FUNCTION_BLOCK TcpConnection
VAR_INPUT
END_VAR
VAR_OUTPUT
END_VAR
VAR
	fbSocketListion : FB_SocketListen;
	fbSocketAccept : FB_SocketAccept;
	fbSocketConnect : FB_SocketConnect;
	fbSocketClose : FB_SocketClose;
	fbSocketCloseAll : FB_SocketCloseAll;
	fbSocketSend : FB_SocketSend;
	fbSocketReceive : FB_SocketReceive;
	fbGetLinkStatus: FB_SocketGetLinkStatus;
	
	CurrentSocket : T_HSOCKET;
	bEstablished : BOOL;
	_HistorySocketIndex : UDINT := 0;
	_HistorySocket : ARRAY[0..HISTORYSOCKET_MAX] OF T_HSOCKET;
	
	ErrorID : UDINT;
	
END_VAR

VAR CONSTANT
	SOCKETEMPTY: T_HSOCKET 
		:= (handle := 0, 
			localAddr := (nPort := 0, sAddr := ''), 
			remoteAddr := (nPort := 0, sAddr := ''));
	HISTORYSOCKET_MAX: UDINT  := 19;
END_VAR

METHOD CheckState : BOOL
VAR_INPUT
END_VAR
fbGetLinkStatus.hSocket := CurrentSocket;
fbGetLinkStatus(bExecute:= TRUE);
IF fbGetLinkStatus.bBusy THEN
	(*Checking*)
ELSE
	IF fbGetLinkStatus.bError OR fbGetLinkStatus.bLinkError THEN
		CheckState := TRUE;
		ErrorID := fbGetLinkStatus.nErrId;
	ELSE
		CheckState := FALSE;
	END_IF
	fbGetLinkStatus(bExecute:= FALSE);
END_IF
END_METHOD

METHOD Close : BOOL
VAR_INPUT
END_VAR
IF CurrentSocket.handle = 0 THEN
	Close := FALSE;
ELSE
	fbSocketClose.hSocket := CurrentSocket;
	fbSocketClose(bExecute := TRUE);
	IF fbSocketClose.bBusy THEN
		(* Closing *)
	ELSE
		IF fbSocketClose.bError THEN
			Close := FALSE;
			ErrorID := fbSocketClose.nErrId;
		ELSE
			Close := TRUE;
		END_IF
		(* Whether the connection is closed or not, clear the CurrentSocket *)
		fbSocketClose(bExecute := FALSE);
		CurrentSocket := SOCKETEMPTY;
	END_IF
END_IF
END_METHOD

METHOD INTERNAL CloseAll : BOOL
VAR_INPUT
END_VAR
fbSocketCloseAll(bExecute:= TRUE);
END_METHOD

METHOD Connect : BOOL
VAR_INPUT
	RemoteIpAddr : T_IPv4Addr;
	RemotePort : UDINT;
END_VAR

VAR

END_VAR
IF CurrentSocket.handle <> 0 THEN
	Connect := TRUE;
	RETURN;
ELSE
	IF RemoteIpAddr = '' OR RemotePort = 0 THEN
		Connect := FALSE;
		RETURN;
	ELSE
		fbSocketConnect.sRemoteHost := RemoteIpAddr;
		fbSocketConnect.nRemotePort := RemotePort;
		fbSocketConnect(bExecute := TRUE);
		IF fbSocketConnect.bBusy THEN
			(* Connecting *)
		ELSE
			IF fbSocketConnect.bError THEN
				fbSocketConnect(bExecute := FALSE);
				Connect := FALSE;
				ErrorID := fbSocketConnect.nErrId;
			ELSE
				fbSocketConnect(bExecute := FALSE);
				CurrentSocket := fbSocketConnect.hSocket;
				(* Store to history array *)
				IF _HistorySocketIndex > HISTORYSOCKET_MAX THEN
					_HistorySocketIndex := 0;
				END_IF
				_HistorySocket[_HistorySocketIndex] := fbSocketConnect.hSocket;
				
			END_IF
		END_IF
	END_IF
END_IF
END_METHOD

PROPERTY ErrID : udint
GET
ErrID := ErrorID;
END_GET
END_PROPERTY

ACTION fbCall:
fbSocketListion(
	sSrvNetId:= , 
	sLocalHost:= , 
	nLocalPort:= , 
	bExecute:= , 
	tTimeout:= , 
	bBusy=> , 
	bError=> , 
	nErrId=> , 
	hListener=> );
fbSocketAccept(
	sSrvNetId:= , 
	hListener:= , 
	bExecute:= , 
	tTimeout:= , 
	bAccepted=> , 
	bBusy=> , 
	bError=> , 
	nErrId=> , 
	hSocket=> );
fbSocketConnect(
	sSrvNetId:= , 
	sRemoteHost:= , 
	nRemotePort:= , 
	bExecute:= , 
	tTimeout:= , 
	bBusy=> , 
	bError=> , 
	nErrId=> , 
	hSocket=> );
fbSocketClose(
	sSrvNetId:= , 
	hSocket:= , 
	bExecute:= , 
	tTimeout:= , 
	bBusy=> , 
	bError=> , 
	nErrId=> );
fbSocketCloseAll(
	sSrvNetId:= , 
	bExecute:= , 
	tTimeout:= , 
	bBusy=> , 
	bError=> , 
	nErrId=> );
fbSocketSend(
	sSrvNetId:= , 
	hSocket:= , 
	cbLen:= , 
	pSrc:= , 
	bExecute:= , 
	tTimeout:= , 
	bBusy=> , 
	bError=> , 
	nErrId=> );
fbSocketReceive(
	sSrvNetId:= , 
	hSocket:= , 
	cbLen:= , 
	pDest:= , 
	bExecute:= , 
	tTimeout:= , 
	bBusy=> , 
	bError=> , 
	nErrId=> , 
	nRecBytes=> );
END_ACTION

PROPERTY hSocket : T_HSOCKET
GET
hSocket := CurrentSocket;
END_GET
END_PROPERTY

METHOD Receive : UDINT
VAR_INPUT
	pData : POINTER TO BYTE;
	nLength : UDINT;
END_VAR
IF pData = 0 OR nLength = 0 THEN
	Receive := 0;
	RETURN;
ELSE
	fbSocketReceive.pDest := pData;
	fbSocketReceive.cbLen := nLength;
	fbSocketReceive.hSocket := CurrentSocket;
	fbSocketReceive(bExecute:= TRUE);
	IF fbSocketReceive.bBusy THEN
		(* Receiving *)
	ELSE
		IF fbSocketReceive.bError THEN
			Receive := 0;
			ErrorID := fbSocketReceive.nErrId;
		ELSE
			Receive := fbSocketReceive.nRecBytes;
		END_IF
		fbSocketReceive(bExecute:= FALSE);
	END_IF
END_IF
END_METHOD

METHOD Send : BOOL
VAR_INPUT
	pData : POINTER TO BYTE;
	nLength : UDINT;
END_VAR
IF pData = 0 OR nLength = 0 THEN
	Send := FALSE;
	RETURN;
ELSE
	fbSocketSend.pSrc := pData;
	fbSocketSend.cbLen := nLength;
	fbSocketSend.hSocket := CurrentSocket;
	fbSocketSend(bExecute:=TRUE);
	IF fbSocketSend.bBusy THEN
		(* Sending *)
	ELSE
		IF fbSocketSend.bError THEN
			Send := FALSE;
			ErrorID := fbSocketSend.nErrId;
		ELSE
			Send := TRUE;
		END_IF
		fbSocketSend(bExecute:=FALSE);
	END_IF
END_IF
END_METHOD

END_FUNCTION_BLOCK

(* stored: Version 1.1.0.1, ProductVersion 3.1.4024.12
   POU TcpConnection: Id {8ab27a36-757a-4cd6-9959-02d6bd57acf3}, SpecialFunc None
   Method CheckState: Id {1bf5cbcd-bb6a-4189-a066-938724933362}
   Method Close: Id {f6e4275e-bfd3-4c63-9d70-832ee22b113e}
   Method CloseAll: Id {905a008b-47b2-49e8-b665-bbe2d02c7168}
   Method Connect: Id {9aaa307b-a96f-477e-b78f-462f241ea09e}
   Property ErrID: Id {902c1ef9-1c9a-45a7-a5f7-930bb7bebdc7}
   Get Get: Id {aa54e7d2-6919-4aef-baa8-36b9563757ff}
   Action fbCall: Id {79d53172-eaa0-4c36-9f34-d5d4765961cf}
   Property hSocket: Id {82fc8d72-48ab-4d32-942d-05670e227e20}
   Get Get: Id {f574aed7-5107-46a4-9eeb-e9c8bed9b464}
   Method Receive: Id {98be8af7-8111-48f7-9d93-c08d968bb4d6}
   Method Send: Id {d4bef882-7da4-41a0-9aef-03df82d24bc9} *)
